// TIA Portal project "Project14" (V19)

(* hardware
DEVICE "S7-1200 station_1"  S7-1200 Station
   slot 0: "Rack_0"  S7-1200 Rack  Rack  V1.0
   slot 1: "PLC_1"  CPU 1211C DC/DC/DC  6ES7 211-1AE40-0XB0  V4.6
   slot 101: "CM 1241 (RS422/485)_1"  6ES7 241-1CH32-0XB0  V2.2
*)

// ===== PLC "PLC_1"  CPU 1211C DC/DC/DC =====

DATA_BLOCK "HOLD_REG_TCP"   // DB3
{ S7_Optimized_Access := 'TRUE' }
VERSION : 0.1
   VAR
      HOLD_REG : Array[0..1] of Int;
      ip : TCON_IP_v4;
   END_VAR
BEGIN
   ip.RemoteAddress.ADDR[1] := 192;
   ip.RemoteAddress.ADDR[2] := 168;
   ip.RemoteAddress.ADDR[3] := 0;
   ip.RemoteAddress.ADDR[4] := 55;
   ip.LocalPort := 502;
END_DATA_BLOCK

FUNCTION_BLOCK "Modbus_Server"   // FB1, LAD
{ S7_Optimized_Access := 'TRUE' }
VERSION : 0.1
BEGIN

REGION Network 1
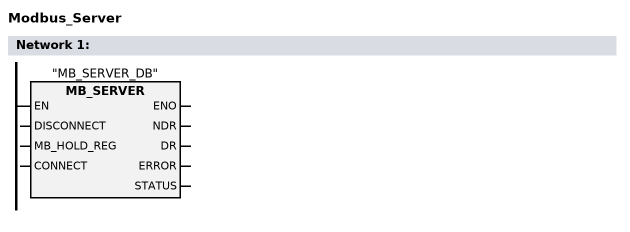
   "MB_SERVER_DB"();   // MB_SERVER
END_REGION
END_FUNCTION_BLOCK

FUNCTION_BLOCK "Modbus_Master"   // FB2, LAD
{ S7_Optimized_Access := 'TRUE' }
VERSION : 0.1
BEGIN

REGION Network 1
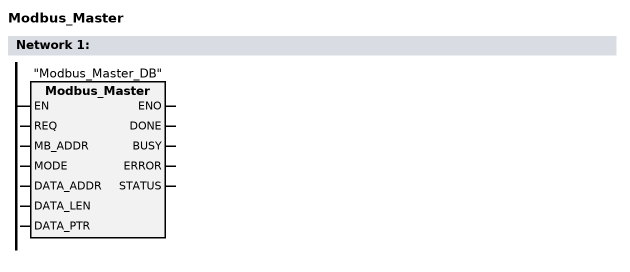
   "Modbus_Master_DB"();   // Modbus_Master
END_REGION
END_FUNCTION_BLOCK

ORGANIZATION_BLOCK "Main"   // OB1, LAD, ProgramCycle
TITLE = "Main Program Sweep (Cycle)"
{ S7_Optimized_Access := 'TRUE' }
VERSION : 0.1
   VAR_INPUT
      Initial_Call : Bool;   // Initial call of this OB
      Remanence : Bool;   // =True, if remanent data are available
   END_VAR
BEGIN
END_ORGANIZATION_BLOCK